{attribute 'qualified_only'}
{attribute 'strict'}
TYPE FeedrateInterpolation :
(
	CONST := Tc2_PlcInterpolation.E_NciFeedRateIpol.E_NciFeedrateIpolConstant,
    LINEAR := Tc2_PlcInterpolation.E_NciFeedRateIpol.E_NciFeedrateIpolLinear
) UINT;
END_TYPE

(* stored: Version 1.1.0.1, ProductVersion 3.1.4024.12
   DUT FeedrateInterpolation: Id {99693232-259d-4d4e-a2eb-f524adca5c8e} *)
